PROGRAM PRG_PF2K2_WFS
VAR
    {attribute 'pytmc' := 'pv: PF2K2:WFS'}
    {attribute 'TcLinkTo' := '.fbThermoCouple1.bError 		:= TIIB[PF2K2-EL3314-E5]^TC Inputs Channel 1^Status^Error;
                              .fbThermoCouple1.bUnderrange	:= TIIB[PF2K2-EL3314-E5]^TC Inputs Channel 1^Status^Underrange;
                              .fbThermoCouple1.bOverrange 	:= TIIB[PF2K2-EL3314-E5]^TC Inputs Channel 1^Status^Overrange;
                              .fbThermoCouple1.iRaw 		:= TIIB[PF2K2-EL3314-E5]^TC Inputs Channel 1^Value;
                              .fbThermoCouple2.bError 		:= TIIB[PF2K2-EL3314-E5]^TC Inputs Channel 2^Status^Error;
                              .fbThermoCouple2.bUnderrange 	:= TIIB[PF2K2-EL3314-E5]^TC Inputs Channel 2^Status^Underrange;
                              .fbThermoCouple2.bOverrange 	:= TIIB[PF2K2-EL3314-E5]^TC Inputs Channel 2^Status^Overrange;
                              .fbThermoCouple2.iRaw 		:= TIIB[PF2K2-EL3314-E5]^TC Inputs Channel 2^Value'}
    fbPF2K2: FB_WFS;

    fbStateSetup: FB_StateSetupHelper;
    stDefault: ST_PositionState := (
        fVelocity := 1,
        bMoveOk := TRUE,
        bValid := TRUE
    );
END_VAR


fbStateSetup(stPositionState:=stDefault, bSetDefault:=TRUE);

fbStateSetup(stPositionState:=fbPF2K2.stOut, fPosition:=-15.00, sPmpsState:='PF2K2:WFS-OUT');
fbStateSetup(stPositionState:=fbPF2K2.stTarget1, fPosition:=-97.789, sPmpsState:='PF2K2:WFS-TARGET1');
fbStateSetup(stPositionState:=fbPF2K2.stTarget2, fPosition:=-83.416, sPmpsState:='PF2K2:WFS-TARGET2');
fbStateSetup(stPositionState:=fbPF2K2.stTarget3, fPosition:=-69.043, sPmpsState:='PF2K2:WFS-TARGET3');
fbStateSetup(stPositionState:=fbPF2K2.stTarget4, fPosition:=-54.669, sPmpsState:='PF2K2:WFS-TARGET4');
fbStateSetup(stPositionState:=fbPF2K2.stTarget5, fPosition:=-40.296, sPmpsState:='PF2K2:WFS-TARGET5');

fbPF2K2(
    fbFFHWO := GVL.fbFastFaultOutput2,
    fbArbiter := GVL.fbArbiter2,
    stYStage := Main.M22,
    stZStage := Main.M23,
    sDeviceName := 'PF2K2:WFS',
    sTransitionKey := 'PF2K2:WFS-TRANSITION',
    bEnableMotion := TRUE,
    bEnableBeamParams := TRUE,
    bEnablePositionLimits := TRUE,
    eEnumGet=>GVL.ePF2K2State,
);

END_PROGRAM

(* stored: Version 1.1.0.1, ProductVersion 3.1.4022.18
   POU PRG_PF2K2_WFS: Id {e443567e-cf8b-49d1-bdca-a5884362d234}, SpecialFunc None *)
